TYPE ST_CartesianPoint :
STRUCT
  x : LREAL;
  y : LREAL;
  z : LREAL;
  a : LREAL;
  b : LREAL;
  c : LREAL;
END_STRUCT
END_TYPE

(* stored: Version 1.1.0.1
   DUT ST_CartesianPoint: Id {03d495c8-b7b1-4578-8869-2eb32cf9188e} *)
